PROGRAM TimeGet
VAR
	NT_GetTime: NT_GetTime;
END_VAR

NT_GetTime(
	NETID:= , 
	START:= , 
	TMOUT:= , 
	BUSY=> , 
	ERR=> , 
	ERRID=> , 
	TIMESTR=> );

END_PROGRAM

(* stored: Version 1.1.0.1, ProductVersion 3.1.4024.0
   POU TimeGet: Id {c59476ad-6469-4aa9-ab3c-361713477fde}, SpecialFunc None *)
